// Device/Application/Zakalka_program
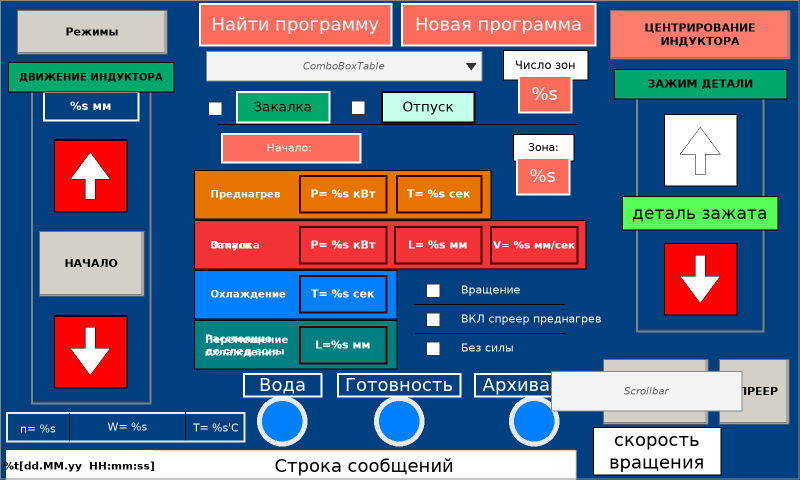
VISUALIZATION Zakalka_program  // 800x480
VAR_IN_OUT
END_VAR
VAR
	bAckSel : BOOL;
	bAckVisible : BOOL;
	bHistory : BOOL;
	bFreezeScrlPos : BOOL;
END_VAR
    RoundedRectangle (194,320 203x49), colour toggle: ZAKALKA.Zakalka_last_zona
    RoundedRectangle (194,170 297x49)
    RoundedRectangle (194,220 392x49)
    RoundedRectangle (194,270 203x49), colour toggle: NOT(ZAKALKA.Zakalka_last_zona), invisible if: ZAKALKA.Zakalka_otpusk_active
    Textfield (513,134 61x27), "Зона:"
    RoundedRectangle (194,270 203x49), invisible if: NOT(ZAKALKA.Zakalka_otpusk_active)
    Textfield (204,279 86x30), "Охлаждение", input disabled if: NOT(ZAKALKA.Zakalka_last_zona)
    Button (603,359 105x65), "ВРАЩЕНИЕ", colour toggle: PLC_PRG.DET_CIRCLE_ON, pressed state: PLC_PRG.DET_CIRCLE_ON
        toggle PLC_PRG.DET_CIRCLE_ON
    Button (719,359 70x65), "СПРЕЕР", colour toggle: PLC_PRG.SPREER_ON, pressed state: PLC_PRG.SPREER_ON
        toggle PLC_PRG.SPREER_ON
    RoundedRectangle (299,275 88x38), "T= %s сек", tooltip "Переменная для отпуска", text variable: GVL.t_freeze[zona_rabochaya+10], invisible if: ZAKALKA.Zakalka_otpusk_active, input disabled if: NOT(ZAKALKA.Zakalka_last_zona)
        OnMouseClick: write GVL.t_freeze[zona_rabochaya+10] via VisuDialogs.Numpad
    Textfield (204,179 91x30), "Преднагрев"
    RoundedRectangle (299,175 88x38), "P= %s кВт", text variable: GVL.P_nachaln_nagrev[zona_rabochaya+10], invisible if: ZAKALKA.Zakalka_otpusk_active
        OnMouseClick: write GVL.P_nachaln_nagrev[zona_rabochaya+10] via VisuDialogs.Numpad, min 1, max 160
    Ellipse (374,396 50x50), colour toggle: GVL.DY_gotovn
    Ellipse (509,396 50x50), colour toggle: Archive.arch_en
    RoundedRectangle (396,175 86x38), "T= %s сек", text variable: GVL.t_nachaln_nagrev[zona_rabochaya+10], invisible if: ZAKALKA.Zakalka_otpusk_active
        OnMouseClick: write GVL.t_nachaln_nagrev[zona_rabochaya+10] via VisuDialogs.Numpad
    Textfield (152,450 424x32), "Строка сообщений", text variable: PLC_PRG.START, text list: 'Warning_Text_list', text index: PLC_PRG.WarningText_mod
    RoundedRectangle (474,373 120x24), "Архивация"
    Button (610,10 180x49), "ЦЕНТРИРОВАНИЕ ИНДУКТОРА"
        OnMouseClick:  Dialog=Center_indukt, OpenModal=True, OpenCentered=True
    Textfield (503,50 85x30), "Число зон"
    RoundedRectangle (518,75 54x38), "%s", text variable: chislo_zon
        OnMouseClick: write chislo_zon via VisuDialogs.Numpad, min 1, max 20
        OnDialogClosed: execute { PLC_PRG.Req_OverWriting_param:=TRUE; PLC_PRG.Req_WR_Params:=FALSE; }
    RoundedRectangle (337,373 124x24), "Готовность"
    RoundedRectangle (636,78 128x254)
    RoundedRectangle (664,243 73x72), colour toggle: PLC_PRG.ZAGIM_DOWN
    RoundedRectangle (664,243 73x72), invisible if: PLC_PRG.in6
        OnMouseUp: execute {  }
    Polygon (680,276) (700,303) (720,276) (705,276) (705,255) (695,255) (695,276), colour toggle: PLC_PRG.ZAGIM_DOWN
    RoundedRectangle (664,114 73x72), colour toggle: PLC_PRG.ZAGIM_UP
    Polygon (680,154) (700,127) (720,154) (705,154) (705,174) (695,174) (695,154), colour toggle: PLC_PRG.ZAGIM_UP
        OnMouseDown: execute {  }
    Textfield (614,69 173x30), "ЗАЖИМ ДЕТАЛИ"
    RoundedRectangle (622,196 156x34), "деталь зажата", invisible if: PLC_PRG.in5
    InvisibleInput (657,108 87x85)
        tap PLC_PRG.ZAGIM_UP
    InvisibleInput (659,238 87x85)
        OnMouseDown: execute { PLC_PRG.ZAGIM_DOWN := TRUE; }
        OnMouseUp: execute { PLC_PRG.ZAGIM_DOWN := FALSE; }
    RoundedRectangle (593,427 128x48), "скорость вращения", colour toggle: NOT(PLC_PRG.in6)
        OnMouseClick: execute {
            IF (PLC_PRG.DET_CIRCLE_SPIN) THEN
            	PLC_PRG.DET_CIRCLE_SPIN := FALSE;
            	ELSE PLC_PRG.DET_CIRCLE_SPIN := TRUE;
            END_IF
        }
    Scrollbar (551,371 191x40), text variable: PLC_PRG.MB_4_20_kanal_2, invisible if: NOT(PLC_PRG.DET_CIRCLE_SPIN)
        p1057716461: PLC_PRG.MB_4_20_kanal_2
    Checkbox (349,93 30x29), variable: ZAKALKA.Otpusk_on
    Rectangle (381,91 94x32), "Отпуск", colour toggle: NOT(ZAKALKA.Zakalka_otpusk_active), input disabled if: NOT(ZAKALKA.Otpusk_on)
        OnMouseDown: execute { ZAKALKA.Zakalka_otpusk_active := FALSE; }
    Rectangle (236,91 94x32), "Закалка", colour toggle: NOT(ZAKALKA.Zakalka_otpusk_active), input disabled if: NOT(ZAKALKA.Zakalka_on)
        OnMouseDown: execute {
            IF ZAKALKA.Otpusk_on THEN
            	ZAKALKA.Zakalka_otpusk_active := TRUE;
            END_IF
        }
    Checkbox (206,94 30x29), variable: ZAKALKA.Zakalka_on
    Textfield (204,230 58x30), "Отпуск", invisible if: ZAKALKA.Zakalka_otpusk_active
    RoundedRectangle (299,226 88x38), "P= %s кВт", tooltip "Переменная для отпуска", text variable: GVL.P_nagrev[zona_rabochaya+10], invisible if: ZAKALKA.Zakalka_otpusk_active
        OnMouseClick: write GVL.P_nagrev[zona_rabochaya+10] via VisuDialogs.Numpad, min 1, max 160
    RoundedRectangle (490,226 88x38), "V= %s мм/сек", tooltip "Переменная для отпуска", text variable: V_peremeshenia[zona_rabochaya+10], invisible if: ZAKALKA.Zakalka_otpusk_active
        OnMouseClick: write GVL.V_peremeshenia[zona_rabochaya+10] via VisuDialogs.Numpad
        OnDialogClosed: execute { PLC_PRG.Req_OverWriting_param:=TRUE; PLC_PRG.Req_WR_Params:=FALSE; }
    RoundedRectangle (394,226 88x38), "L= %s мм", tooltip "Переменная для отпуска", text variable: L_peremeshenia[zona_rabochaya+10], invisible if: ZAKALKA.Zakalka_otpusk_active
        OnMouseClick: write GVL.L_peremeshenia[zona_rabochaya+10] via VisuDialogs.Numpad
        OnDialogClosed: execute { PLC_PRG.Req_OverWriting_param:=TRUE; PLC_PRG.Req_WR_Params:=FALSE; }
    RoundedRectangle (221,133 140x30), "Начало:", text list: 'NachaloVerhNiz', text index: ZAKALKA.zakalka_nachalo
        OnMouseClick: execute {
            IF ZAKALKA.zakalka_nachalo = 0 THEN
            	ZAKALKA.zakalka_nachalo := 1;
            ELSE
            	ZAKALKA.zakalka_nachalo := 0;
            END_IF
            PLC_PRG.Req_OverWriting_param:=TRUE;
            PLC_PRG.Req_WR_Params:=FALSE;
        }
    Textfield (202,330 96x30), "Расстояние до след зоны", invisible if: ZAKALKA.Zakalka_last_zona
    RoundedRectangle (299,326 88x38), "L=%s мм", tooltip "Переменная для отпуска", text variable: L_to_next_zone[zona_rabochaya+1], invisible if: ZAKALKA.Zakalka_last_zona
        OnMouseClick: write L_to_next_zone[zona_rabochaya+1] via VisuDialogs.Numpad
        OnDialogClosed: execute { PLC_PRG.Req_OverWriting_param:=TRUE; PLC_PRG.Req_WR_Params:=FALSE; }
    RoundedRectangle (31,75 120x329)
    RoundedRectangle (54,315 73x72), colour toggle: PLC_PRG.Butt_DOWN
    RoundedRectangle (54,316 73x72), invisible if: PLC_PRG.in3
        OnMouseUp: execute {  }
    Polygon (70,348) (90,375) (110,348) (95,348) (95,327) (85,327) (85,348), colour toggle: PLC_PRG.Butt_DOWN
        OnMouseDown: execute {  }
    InvisibleInput (49,310 85x82)
        OnMouseDown: execute { PLC_PRG.UP_DOWN := 2; PLC_PRG.Butt_DOWN := TRUE; }
        OnMouseUp: execute { PLC_PRG.UP_DOWN := 0; PLC_PRG.Butt_DOWN := FALSE; }
    RoundedRectangle (54,139 73x72), colour toggle: PLC_PRG.Butt_UP
        OnMouseUp: execute {  }
    RoundedRectangle (54,140 73x72), invisible if: PLC_PRG.in6
    Polygon (70,179) (90,152) (110,179) (95,179) (95,199) (85,199) (85,179), colour toggle: PLC_PRG.Butt_UP
        OnMouseDown: execute {  }
    InvisibleInput (49,135 85x82)
        OnMouseDown: execute { PLC_PRG.UP_DOWN := 1; PLC_PRG.Butt_UP := TRUE; }
        OnMouseUp: execute { PLC_PRG.UP_DOWN := 0; PLC_PRG.Butt_UP := FALSE; }
    Textfield (43,91 96x30), "%s мм", text variable: tekyheePosition_lcd
    Textfield (8,62 166x30), "ДВИЖЕНИЕ ИНДУКТОРА"
    Textfield (6,450 147x32), "%t[dd.MM.yy HH:mm:ss]"
    Rectangle (6,412 239x30)
    Line (69,413) (69,441)
    Textfield (8,419 60x20), "n= %s", text variable: n_nagrev
    Line (185,412) (185,440)
    Textfield (71,417 113x20), "W= %s", text variable: W_schet_vat
    Textfield (186,418 60x20), "T= %s'C", text variable: T_rad_max
    RoundedRectangle (401,3 195x43), "Новая программа"
        OnMouseClick: write ZAKALKA.new_prog via KeypadNumpad
        OnMouseClick: execute { ZAKALKA.pressed_create_new_prog:=true; }
    RoundedRectangle (199,3 193x43), "Найти программу"
        OnMouseClick: write ZAKALKA.SearchThroughArray via KeypadNumpad
        OnMouseClick: execute {
            ZAKALKA.pressed_find_prog:=TRUE;
            ZAKALKA.i_result_prog:=2;
            ZAKALKA.enter_prog:=2;
        }
    ComboBoxTable (206,51 276x30), variable: ZAKALKA.enter_prog, data array: ZAKALKA.result_prog
        p1128707560: ZAKALKA.i_result_prog
        p3854506369: ZAKALKA.result_prog[INDEX]
    Textfield (204,279 86x30), "Охлаждение", invisible if: NOT(ZAKALKA.Zakalka_otpusk_active)
    RoundedRectangle (299,275 88x38), "T= %s сек", tooltip "Переменная для закалки", text variable: t_freeze[zona_rabochaya], invisible if: NOT(ZAKALKA.Zakalka_otpusk_active)
        OnMouseClick: write t_freeze[zona_rabochaya] via VisuDialogs.Numpad
        OnDialogClosed: execute { PLC_PRG.Req_OverWriting_param:=TRUE; PLC_PRG.Req_WR_Params:=FALSE; }
    RoundedRectangle (299,175 88x38), "P= %s кВт", tooltip "Переменная для отпуска", text variable: P_nachaln_nagrev[zona_rabochaya], invisible if: NOT(ZAKALKA.Zakalka_otpusk_active)
        OnMouseClick: write P_nachaln_nagrev[zona_rabochaya] via VisuDialogs.Numpad, min 1, max 160
        OnDialogClosed: execute { PLC_PRG.Req_OverWriting_param:=TRUE; PLC_PRG.Req_WR_Params:=FALSE; }
    RoundedRectangle (396,175 86x38), "T= %s сек", tooltip "Переменная для отпуска", text variable: t_nachaln_nagrev[zona_rabochaya], invisible if: NOT(ZAKALKA.Zakalka_otpusk_active)
        OnMouseClick: write t_nachaln_nagrev[zona_rabochaya] via VisuDialogs.Numpad
        OnDialogClosed: execute { PLC_PRG.Req_OverWriting_param:=TRUE; PLC_PRG.Req_WR_Params:=FALSE; }
    Textfield (204,230 58x30), "Закалка", invisible if: NOT(ZAKALKA.Zakalka_otpusk_active)
    RoundedRectangle (299,226 88x38), "P= %s кВт", tooltip "Переменная для закалки", text variable: P_nagrev[zona_rabochaya], invisible if: NOT(ZAKALKA.Zakalka_otpusk_active)
        OnMouseClick: write P_nagrev[zona_rabochaya] via VisuDialogs.Numpad, min 1, max 160
        OnDialogClosed: execute { PLC_PRG.Req_OverWriting_param:=TRUE; PLC_PRG.Req_WR_Params:=FALSE; }
    RoundedRectangle (490,226 88x38), "V= %s мм/сек", tooltip "Переменная для закалки", text variable: V_peremeshenia[zona_rabochaya], invisible if: NOT(ZAKALKA.Zakalka_otpusk_active)
        OnMouseClick: write V_peremeshenia[zona_rabochaya] via VisuDialogs.Numpad
        OnDialogClosed: execute { PLC_PRG.Req_OverWriting_param:=TRUE; PLC_PRG.Req_WR_Params:=FALSE; }
    RoundedRectangle (394,226 88x38), "L= %s мм", tooltip "Переменная для закалки", text variable: L_peremeshenia[zona_rabochaya], invisible if: NOT(ZAKALKA.Zakalka_otpusk_active)
        OnMouseClick: write L_peremeshenia[zona_rabochaya] via VisuDialogs.Numpad
        OnDialogClosed: execute { PLC_PRG.Req_OverWriting_param:=TRUE; PLC_PRG.Req_WR_Params:=FALSE; }
    Button (17,10 150x44), "Режимы"
        OnMouseClick:  Assign=Regim_choice, Type=Assignment
    Ellipse (257,396 50x50), colour toggle: PLC_PRG.in1
    RoundedRectangle (243,373 79x24), "Вода"
    Button (39,231 105x65), "НАЧАЛО", colour toggle: PLC_PRG.DY_kn_nachalo, pressed state: PLC_PRG.DY_kn_nachalo
        toggle PLC_PRG.DY_kn_nachalo
        OnMouseClick: execute { PLC_PRG.Req_OverWriting_param:=TRUE; PLC_PRG.Req_WR_Params:=FALSE; }
    RoundedRectangle (516,157 54x38), "%s", text variable: zona_rabochaya
        OnMouseClick: write zona_rabochaya via VisuDialogs.Numpad, min 1, max GVL.chislo_zon
    Line (217,124) (578,124)
    Checkbox (424,276 30x29), tooltip "Включить вращение", variable: ZAKALKA.rotation_on
    Checkbox (424,305 30x29), variable: ZAKALKA.spreer_prednagrev
    Checkbox (424,334 30x29), variable: ZAKALKA.diagnostik
    Textfield (458,280 76x20), "Вращение"
    Textfield (458,309 163x20), "ВКЛ спреер преднагрев"
    Textfield (458,338 94x20), "Без силы"
    Line (414,304) (564,304)
    Line (415,333) (565,333)
    Textfield (202,331 96x30), "Перемещение охлаждения", invisible if: NOT(ZAKALKA.Zakalka_last_zona)
    RoundedRectangle (299,326 88x38), "L=%s мм", tooltip "Переменная для закалки", text variable: ZAKALKA.dy_L_dvig_ohl, invisible if: NOT(ZAKALKA.Zakalka_last_zona)
        OnMouseClick: write ZAKALKA.dy_L_dvig_ohl via VisuDialogs.Numpad
        OnDialogClosed: execute { PLC_PRG.Req_OverWriting_param:=TRUE; PLC_PRG.Req_WR_Params:=FALSE; }
END_VISUALIZATION

// Device/Application/Zakalka_work
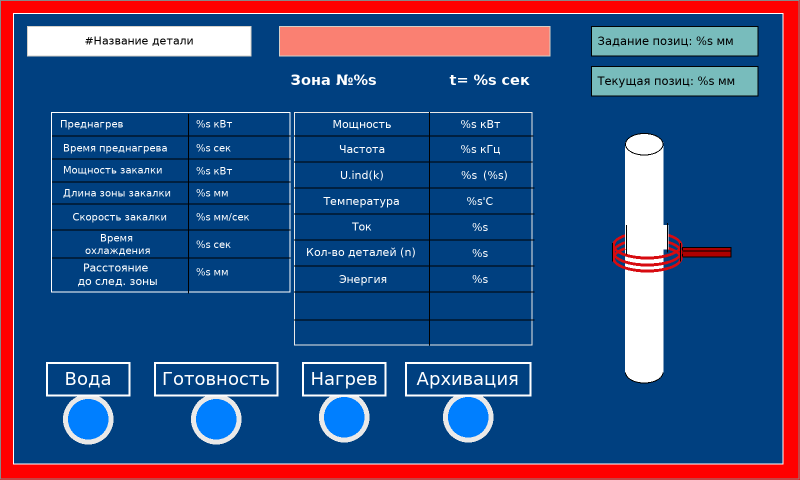
VISUALIZATION Zakalka_work  // 800x480
    Rectangle (13,13 770x451)
    Textfield (279,66 109x28), "Зона №%s", text variable: zona
    Textfield (430,66 120x28), "t= %s сек", text variable: t_prog_LCD
    Textfield (279,26 271x30), text list: 'Status_v_Rabote', text index: GVL.i_t_regim, colour variable: ZAKALKA.color_indukt
    Textfield (591,26 167x30), "Задание позиц: %s мм", text variable: zadachaPosition_lcd
    Textfield (591,66 167x30), "Текущая позиц: %s мм", text variable: tekyheePosition_lcd
    Rectangle (51,112 239x180)
    Line (290,136) (52,136)
    Line (290,159) (52,159)
    Line (290,182) (52,182)
    Line (290,204) (52,204)
    Line (290,230) (52,230)
    Line (188,114) (188,293)
    Textfield (57,160 123x20), "Мощность закалки"
    Textfield (57,183 123x20), "Длина зоны закалки"
    Textfield (57,114 119x20), "Преднагрев"
    Textfield (57,138 122x20), "Время преднагрева"
    Textfield (57,232 122x25), "Время охлаждения"
    Textfield (57,207 126x20), "Скорость закалки"
    Textfield (53,260 129x29), "Расстояние до след. зоны", text variable: zona_rabochaya+1, invisible if: ZAKALKA.L_between_stels
    Textfield (193,114 90x20), "%s кВт", text variable: P_nachaln_nagrev[zona+ZAKALKA.shift_otpusk]
    Textfield (193,183 89x20), "%s мм", text variable: L_peremeshenia[zona+ZAKALKA.shift_otpusk]
    Textfield (193,138 90x20), "%s сек", text variable: t_nachaln_nagrev[zona+ZAKALKA.shift_otpusk]
    Textfield (193,232 90x25), "%s сек", text variable: t_freeze[zona+ZAKALKA.shift_otpusk]
    Textfield (193,207 90x20), "%s мм/сек", text variable: V_peremeshenia[zona+ZAKALKA.shift_otpusk]
    Textfield (193,161 90x20), "%s кВт", text variable: P_nagrev[zona+ZAKALKA.shift_otpusk]
    Textfield (193,262 89x20), "%s мм", text variable: L_to_next_zone[zona+1+ZAKALKA.shift_otpusk], invisible if: ZAKALKA.L_between_stels
    Line (290,258) (52,258)
    Group (625,133 43x290)
        Ellipse (0,228 38x22)
        Rectangle (0,9 38x230)
        Ellipse (0,0 38x22)
    Rectangle (682,247 49x10)
    Line (731,251) (680,251)
    Ellipse (612,231 70x28)
        p3450524324: ZAKALKA.color_indukt
    Ellipse (612,238 70x28)
        p3450524324: ZAKALKA.color_indukt
    Ellipse (612,244 70x28)
        p3450524324: ZAKALKA.color_indukt
    Rectangle (625,225 43x24)
    Line (680,243) (680,261)
        p2175578022: ZAKALKA.color_indukt
    Line (612,243) (612,261)
        p2175578022: ZAKALKA.color_indukt
    Line (667,223) (667,252)
    Line (626,225) (626,254)
    Textfield (27,26 224x30), "#Название детали"
    Rectangle (294,112 238x233)
    Textfield (438,115 85x19), "%s кВт", text variable: P_ind/10
    Textfield (438,140 85x19), "%s кГц", text variable: Frec_LCD_point/10
    Textfield (325,115 74x19), "Мощность"
    Textfield (330,140 64x19), "Частота"
    Line (533,136) (294,136)
    Line (532,162) (294,162)
    Line (534,188) (294,188)
    Textfield (336,166 52x19), "U.ind(k)"
    Textfield (319,192 85x19), "Температура"
    Textfield (450,192 60x19), "%s'C", text variable: T_rad_max
    Line (534,214) (294,214)
    Line (534,240) (294,240)
    Textfield (423,166 57x19), "%s", text variable: U_pit_max
    Line (429,112) (429,345)
    Textfield (316,217 92x20), "Ток"
    Textfield (317,270 92x19), "Энергия"
    Textfield (299,243 124x19), "Кол-во деталей (n)"
    Ellipse (191,394 50x50), colour toggle: GVL.DY_gotovn
    Ellipse (443,392 50x50), colour toggle: Archive.arch_en
    Ellipse (63,394 50x50), colour toggle: PLC_PRG.in1
    Ellipse (319,392 50x50), colour toggle: PLC_PRG.START
    Line (534,266) (294,266)
    Line (534,292) (294,292)
    Line (534,320) (294,320)
    Textfield (432,218 96x19), "%s", text variable: I_lcd
    Textfield (432,244 96x19), "%s", text variable: n_nagrev
    Textfield (432,270 96x19), "%s", text variable: W_schet_vat
    Textfield (480,166 48x19), "(%s)", text variable: zona_reg
    RoundedRectangle (405,362 126x34), "Архивация"
    RoundedRectangle (46,362 84x34), "Вода"
    RoundedRectangle (154,362 124x34), "Готовность"
    RoundedRectangle (302,362 84x34), "Нагрев"
END_VISUALIZATION

(* text list Modbus_Error_list (id | default)
  0 | Связь есть
  1 | Принятый код функции не может быть обработан
  2 | Адрес данных, указанный в запросе, недоступен
  3 | Значение, содержащееся в поле данных запроса, является недопустимой величиной
  4 | Невосстанавливаемая ошибка имела место, пока ведомое устройство пыталось выполнить затребованное действие
  5 | Ведомое устройство приняло запрос и обрабатывает его, но это требует много времени
  6 | Ведомое устройство занято обработкой команды
  7 | Ведомое устройство при чтении расширенной памяти обнаружило ошибку паритета
  10 | Special error when using devices behind a gateway (Gateway misconfigured/busy)
  11 | Special error when using devices behind a gateway (Device does not respond)
  161 | There was no response in time
  162 | The checksum of the response is not correct
  163 | The response is not from the expected Slave
  164 | The response is not the expected function code
  165 | Local COM Port error. Request was not sent
   |  *)

(* text list Status_v_Rabote (id | default)
  0 | Преднагрев
  1 | Закалка
  2 | Охлаждение
  3 | 
  4 | Движение на позицию
   |  *)

(* text list Warning_Text_list (id | default)
  1 | Нет питания
  2 | Время закончено
  3 | Высокая температура
  4 | Обрыв датчика температуры
  5 | Ошибка исход механ
  6 | Нет нагрева заготовки
  7 | Сбой резонанса
  8 | Частота больше нормы
  9 | Частота меньше нормы
  10 | Нет воды
  155 | Нет связи
  11 | защита LCD
  12 | защита по току 1
  13 | защита по току 2
  14 | защита по току 3
  15 | защита по току 4
  16 | защита драйвера 1
  17 | защита драйвера 2
  18 | защита драйвера 3
  19 | защита драйвера 4
  20 | Защита всп питание 1
  21 | Защита всп питание 2
  22 | Защита всп питание 3
  23 | Защита всп питание 4
  24 | перегрев радиатора 4
  25 | перегрев радиатора 1
  26 | перегрев радиатора 2
  27 | перегрев радиатора 3
  28 | нет силового питания 4
  29 | нет силового питания 1
  30 | нет силового питания 2
  31 | нет силового питания 3
  32 | перегрев БС
  33 | Ручной режим
  34 | Автомат по мощности
  35 | Пустой индуктор
  36 | нет питания БС
  37 | Закончен автоцикл
  38 | Диагностика
  39 | Автомат по температуре
  40 | Режим не активен
  41 | Блок реж 0 Сбой памяти
  42 | Автомат по температуре
  43 | Автомат по температуре
  44 | Автомат Сушка
  45 | Выбор действия
  46 | Т2 достигнута
  47 | Стоп нагрев
  48 | Охлаждение вода
  49 | Защита платы питания 1
  50 | Защита платы питания 2
  51 | Защита платы питания 3
  52 | Защита платы питания 4
  53 | Стоп авария
  54 | Стоп конвейер
  55 | Подача авария
  56 | Подача заготовки
  57 | Повторный нагрев
  58 | Блокировка режимов 2
  59 | Блокировка режимов 3
  60 | Блокировка режимов 4
  61 | Блокировка режимов 5
  62 | Блокировка режимов 6
  63 | Блокировка режимов 7
  64 | Вход - нет заготовки
  65 | Термоциклирование
  66 | Перегрев заготовки
  67 | Нет заготовки
  68 | Авария механики
  69 | Включено силовое питание
  70 | Переключение постов
  71 | Защита по току 
  72 | Защита по току 5
  73 | Защита по току 6
  74 | Защита по току 7
  75 | Защита по току 8
  76 | Защита драйвера 
  77 | Защита драйвера 5
  78 | Защита драйвера 6
  79 | Защита драйвера 7
  80 | Защита драйвера 8
  81 | Защита тест питания 
  82 | Защита тест питания 5
  83 | Защита тест питания 6
  84 | Защита тест питания 7
  85 | Защита тест питания 8
  86 | Защита U инвертора 
  87 | Защита U инвертора 1
  88 | Защита U инвертора 2
  89 | Защита U инвертора 3
  90 | Защита U инвертора 4
  91 | Защита U инвертора 5
  92 | Защита U инвертора 6
  93 | Защита U инвертора 7
  94 | Защита U инвертора 8
  95 | Нет силового питания 1
  96 | Нет силового питания 2
  97 | Нет силового питания 3
  98 | Нет силового питания 4
  99 | Нет силового питания 5
  100 | Нет силового питания 6
  101 | Нет силового питания 7
  102 | Нет силового питания 8
  103 | Защита пллаты питания 5
  104 | Защита пллаты питания 6
  105 | Защита пллаты питания 7
  106 | Защита пллаты питания 8
  107 | Ошибка драйвер 1
  108 | Ошибка драйвер 2
  109 | Ошибка драйвер 3
  110 | Ошибка драйвер 4
  111 | Ошибка драйвер 5
  112 | Ошибка драйвер 6
  113 | Ошибка драйвер 7
  114 | Ошибка драйвер 8
  115 | Ошибка блока защит
  116 | Защита драйвера 1 старт
  117 | Защита драйвера 2 старт
  118 | Защита драйвера 3 старт
  119 | Защита драйвера 4 старт
  120 | Защита драйвера 5 старт
  121 | Защита драйвера 6 старт
  122 | Защита драйвера 7 старт
  123 | Защита драйвера 8 старт
  124 | Защита тока 1 старт
  125 | Защита тока 2 старт
  126 | Защита тока 3 старт
  127 | Защита тока 4 старт
  128 | Защита тока 5 старт
  129 | Защита тока 6 старт
  130 | Защита тока 7 старт
  131 | Защита тока 8 старт
  132 | Сделать позицию
  133 | Движение на позицию
  134 | Нет этапа нагрева
  135 | Перегрв радиатора 1
  136 | Перегрв радиатора 2
  137 | Перегрв радиатора 3
  138 | Перегрв радиатора 4
  139 | Перегрв радиатора 5
  140 | Перегрв радиатора 6
  141 | Перегрв радиатора 7
  142 | Перегрв радиатора 8
  143 | Обрыв датчика температуры 1
  144 | Обрыв датчика температуры 2
  145 | Обрыв датчика температуры 3
  146 | Обрыв датчика температуры 4
  147 | Обрыв датчика температуры 5
  148 | Обрыв датчика температуры 6
  149 | Обрыв датчика температуры 7
  150 | Обрыв датчика температуры  8
  151 | Перегрев объекта
  152 | Нет воды в спреере
  153 | Ошибка памяти контроллера
  154 | Подъем лотка
  184 | 
  156 | Установка в работе
   |  *)

(* text list NachaloVerhNiz (id | default)
  1 | Начало: ВЕРХ
  0 | Начало: НИЗ
   |  *)
